(*
A list implementation for managing `I_Arg`.  
*)
INTERFACE I_ArgList EXTENDS I_Debug

(*
Provides the maximum capacity of the list.
*)
PROPERTY Cap : UDINT
GET
END_GET
END_PROPERTY

(*
Retrieves the `I_Arg` at the specified index.  
Returns:
- `Ok` - Successfully retrieves the `I_Arg`.
- `Err.Idx` - The list is empty.
- `Err.Ovf` - The specified index is out of bounds.
*)
METHOD Get : Result
VAR_INPUT
	nIndex		: UDINT;
END_VAR
VAR_OUTPUT
	iArg		: I_Arg;
END_VAR
END_METHOD

(*
Returns the current number of elements in the list.
*)
PROPERTY Length : UDINT
GET
END_GET
END_PROPERTY

END_INTERFACE

(* stored: Version 1.1.0.1
   Itf I_ArgList: Id {e91fb910-5bc2-4619-a29f-96e93d2b0a10}
   Property Cap: Id {4edf4f66-c012-4092-a8bf-0f0119e455bf}
   Get Get: Id {815a00dc-b365-44b6-bb0a-997eb63d1d50}
   Method Get: Id {42042ace-be5b-46c2-98b0-007a36c24259}
   Property Length: Id {3405a074-7d0f-4436-8bfa-2cf6a1a1b0ee}
   Get Get: Id {7e0490c5-d846-48c8-8411-2ce39122c896} *)
